% RSLogix 500 project IDENTIFICACION_BAK249.RSS, saved by version 7.30.00.17 %
PROJECT "UNTITLED"    % processor: MicroLogix 1500 %

PROGRAM FILES
  LAD 2 "PRINCIPAL"  5 rungs
  LAD 3 "FLUJO"  5 rungs
  LAD 4 "NIVEL"  9 rungs
  LAD 5 "BOMBAS"  5 rungs
  LAD 6 "FILTROS"  39 rungs

DATA FILES
  O0 OUTPUT  41 elements
  I1 INPUT  59 elements
  S2 STATUS  66 elements
  B3 BINARY  1 elements
  T4 TIMER  3 elements
  C5 COUNTER  1 elements
  R6 CONTROL  12 elements
  N7 INTEGER  84 elements
  F8 FLOAT  30 elements

LADDER 2 "PRINCIPAL"
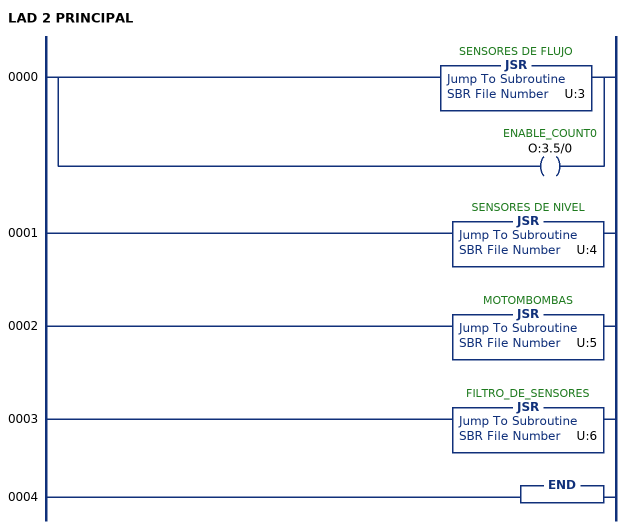
% Rung: 0 %
SOR BST JSR U:3 NXB OTE O:3.5/0 BND EOR
%   U:3  "SENSORES DE FLUJO" %
%   O:3.5/0  ENABLE_COUNT0 %
% Rung: 1 %
SOR JSR U:4 EOR
%   U:4  "SENSORES DE NIVEL" %
% Rung: 2 %
SOR JSR U:5 EOR
%   U:5  "MOTOMBOMBAS" %
% Rung: 3 %
SOR JSR U:6 EOR
%   U:6  FILTRO_DE_SENSORES %
% Rung: 4 %
SOR END EOR

LADDER 3 "FLUJO"
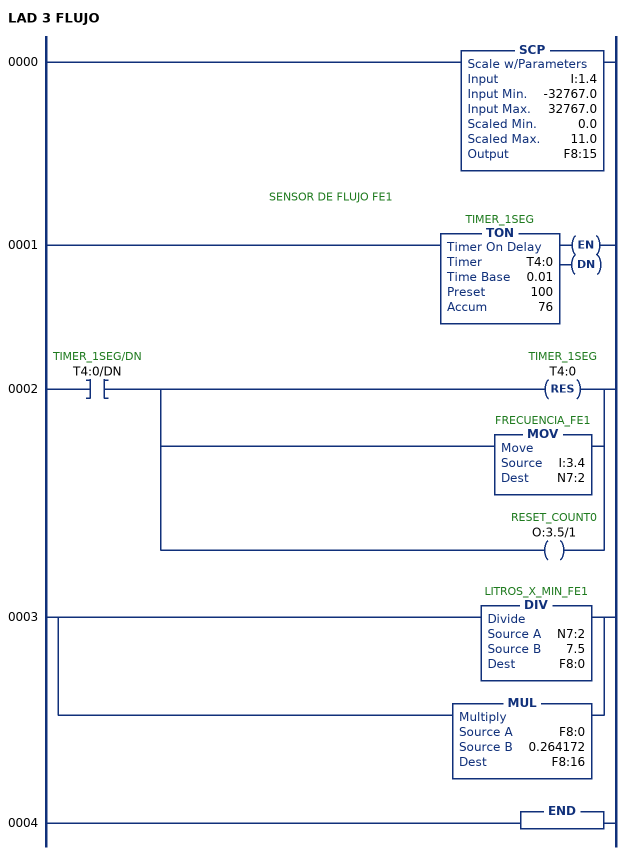
% Rung: 0 %
SOR SCP I:1.4 -32767.0 32767.0 0.0 11.0 F8:15 EOR
%   I:1.4  TRANSMISOR_FIT %
% Rung: 1 %
% SENSOR DE FLUJO FE1 %
SOR TON T4:0 0.01 100 76 EOR
%   T4:0  TIMER_1SEG %
% Rung: 2 %
SOR XIC T4:0/DN BST RES T4:0 NXB MOV I:3.4 N7:2 NXB OTE O:3.5/1 BND EOR
%   T4:0  TIMER_1SEG %
%   N7:2  FRECUENCIA_FE1 %
%   O:3.5/1  RESET_COUNT0 %
% Rung: 3 %
SOR BST DIV N7:2 7.5 F8:0 NXB MUL F8:0 0.264172 F8:16 BND EOR
%   N7:2  FRECUENCIA_FE1 %
%   F8:0  LITROS_X_MIN_FE1 %
% Rung: 4 %
SOR END EOR

LADDER 4 "NIVEL"
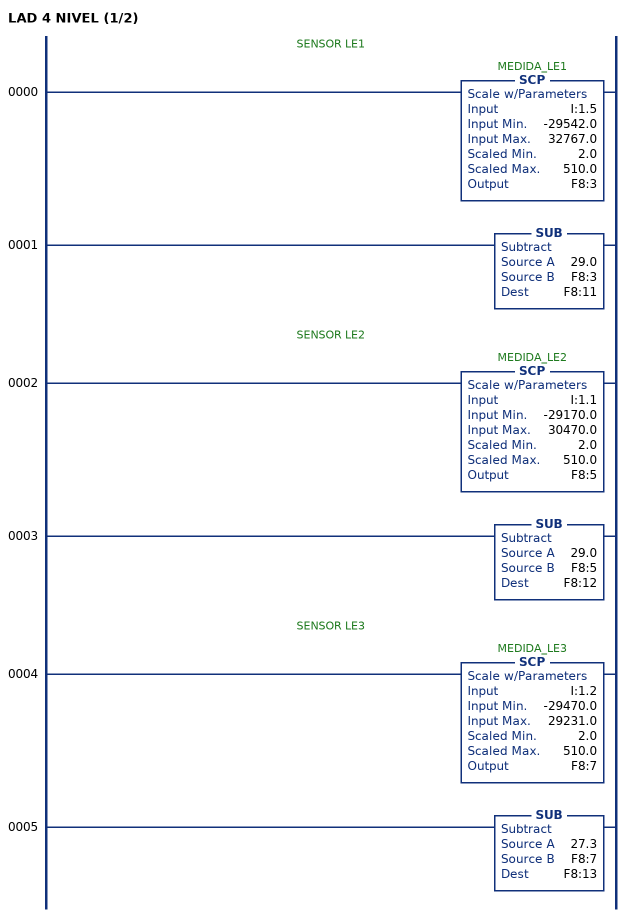
% Rung: 0 %
% SENSOR LE1 %
SOR SCP I:1.5 -29542.0 32767.0 2.0 510.0 F8:3 EOR
%   I:1.5  LE1 %
%   F8:3  MEDIDA_LE1 %
% Rung: 1 %
SOR SUB 29.0 F8:3 F8:11 EOR
%   F8:3  MEDIDA_LE1 %
% Rung: 2 %
% SENSOR LE2 %
SOR SCP I:1.1 -29170.0 30470.0 2.0 510.0 F8:5 EOR
%   I:1.1  LE2 %
%   F8:5  MEDIDA_LE2 %
% Rung: 3 %
SOR SUB 29.0 F8:5 F8:12 EOR
%   F8:5  MEDIDA_LE2 %
% Rung: 4 %
% SENSOR LE3 %
SOR SCP I:1.2 -29470.0 29231.0 2.0 510.0 F8:7 EOR
%   I:1.2  LE3 %
%   F8:7  MEDIDA_LE3 %
% Rung: 5 %
SOR SUB 27.3 F8:7 F8:13 EOR
%   F8:7  MEDIDA_LE3 %

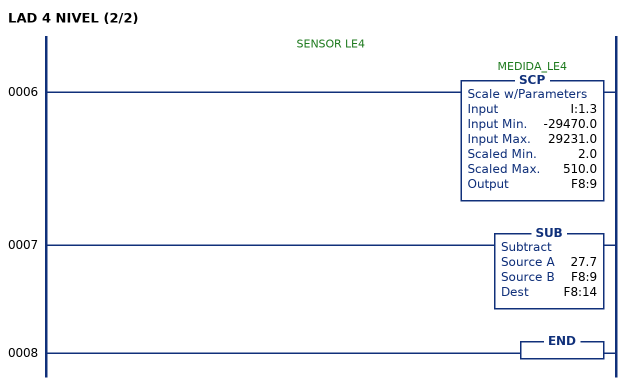
% Rung: 6 %
% SENSOR LE4 %
SOR SCP I:1.3 -29470.0 29231.0 2.0 510.0 F8:9 EOR
%   I:1.3  LE4 %
%   F8:9  MEDIDA_LE4 %
% Rung: 7 %
SOR SUB 27.7 F8:9 F8:14 EOR
%   F8:9  MEDIDA_LE4 %
% Rung: 8 %
SOR END EOR

LADDER 5 "BOMBAS"
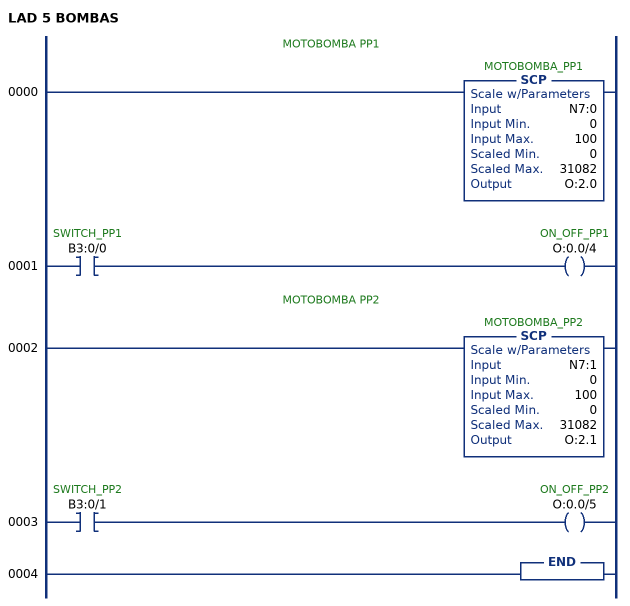
% Rung: 0 %
% MOTOBOMBA PP1 %
SOR SCP N7:0 0 100 0 31082 O:2.0 EOR
%   N7:0  FRECUENCIA_PP1 %
%   O:2.0  MOTOBOMBA_PP1 %
% Rung: 1 %
SOR XIC B3:0/0 OTE O:0.0/4 EOR
%   B3:0/0  SWITCH_PP1 %
%   O:0.0/4  ON_OFF_PP1 %
% Rung: 2 %
% MOTOBOMBA PP2 %
SOR SCP N7:1 0 100 0 31082 O:2.1 EOR
%   O:2.1  MOTOBOMBA_PP2 %
% Rung: 3 %
SOR XIC B3:0/1 OTE O:0.0/5 EOR
%   B3:0/1  SWITCH_PP2 %
%   O:0.0/5  ON_OFF_PP2 %
% Rung: 4 %
SOR END EOR

LADDER 6 "FILTROS"
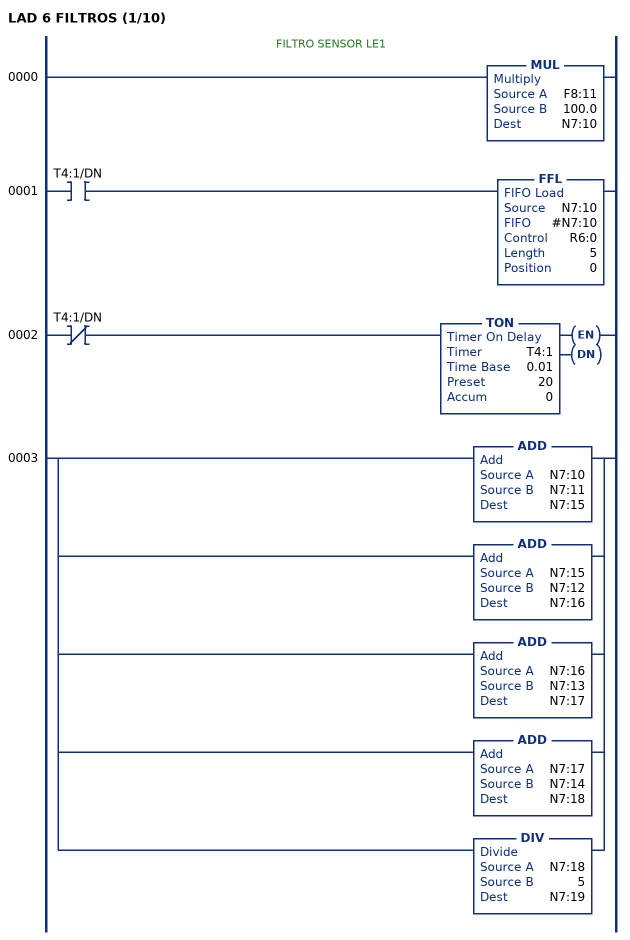
% Rung: 0 %
% FILTRO SENSOR LE1 %
SOR MUL F8:11 100.0 N7:10 EOR
% Rung: 1 %
SOR XIC T4:1/DN FFL N7:10 #N7:10 R6:0 5 0 EOR
% Rung: 2 %
SOR XIO T4:1/DN TON T4:1 0.01 20 0 EOR
% Rung: 3 %
SOR BST ADD N7:10 N7:11 N7:15 NXB ADD N7:15 N7:12 N7:16 NXB ADD N7:16 N7:13 N7:17 NXB ADD N7:17 N7:14 N7:18 NXB DIV N7:18 5 N7:19 BND EOR

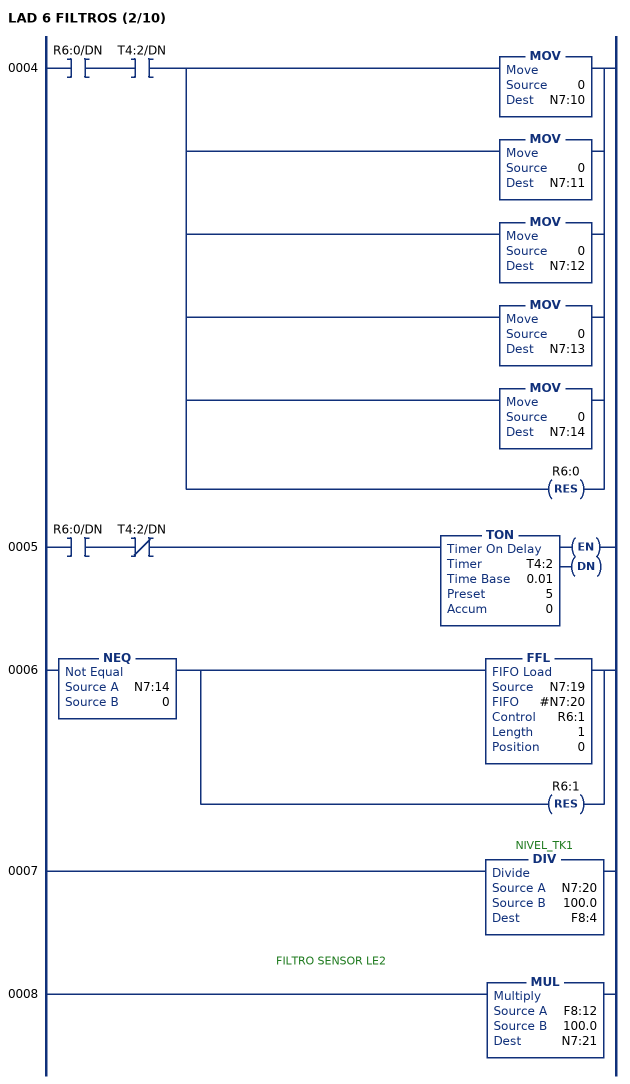
% Rung: 4 %
SOR XIC R6:0/DN XIC T4:2/DN BST MOV 0 N7:10 NXB MOV 0 N7:11 NXB MOV 0 N7:12 NXB MOV 0 N7:13 NXB MOV 0 N7:14 NXB RES R6:0 BND EOR
% Rung: 5 %
SOR XIC R6:0/DN XIO T4:2/DN TON T4:2 0.01 5 0 EOR
% Rung: 6 %
SOR NEQ N7:14 0 BST FFL N7:19 #N7:20 R6:1 1 0 NXB RES R6:1 BND EOR
% Rung: 7 %
SOR DIV N7:20 100.0 F8:4 EOR
%   F8:4  NIVEL_TK1 %
% Rung: 8 %
% FILTRO SENSOR LE2 %
SOR MUL F8:12 100.0 N7:21 EOR

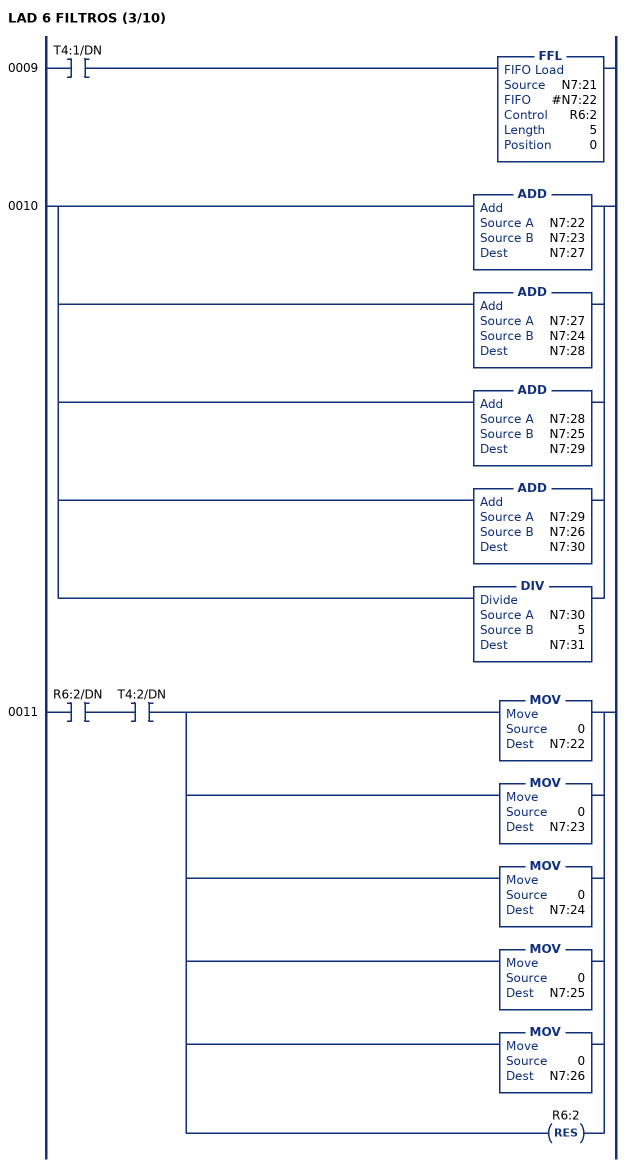
% Rung: 9 %
SOR XIC T4:1/DN FFL N7:21 #N7:22 R6:2 5 0 EOR
% Rung: 10 %
SOR BST ADD N7:22 N7:23 N7:27 NXB ADD N7:27 N7:24 N7:28 NXB ADD N7:28 N7:25 N7:29 NXB ADD N7:29 N7:26 N7:30 NXB DIV N7:30 5 N7:31 BND EOR
% Rung: 11 %
SOR XIC R6:2/DN XIC T4:2/DN BST MOV 0 N7:22 NXB MOV 0 N7:23 NXB MOV 0 N7:24 NXB MOV 0 N7:25 NXB MOV 0 N7:26 NXB RES R6:2 BND EOR

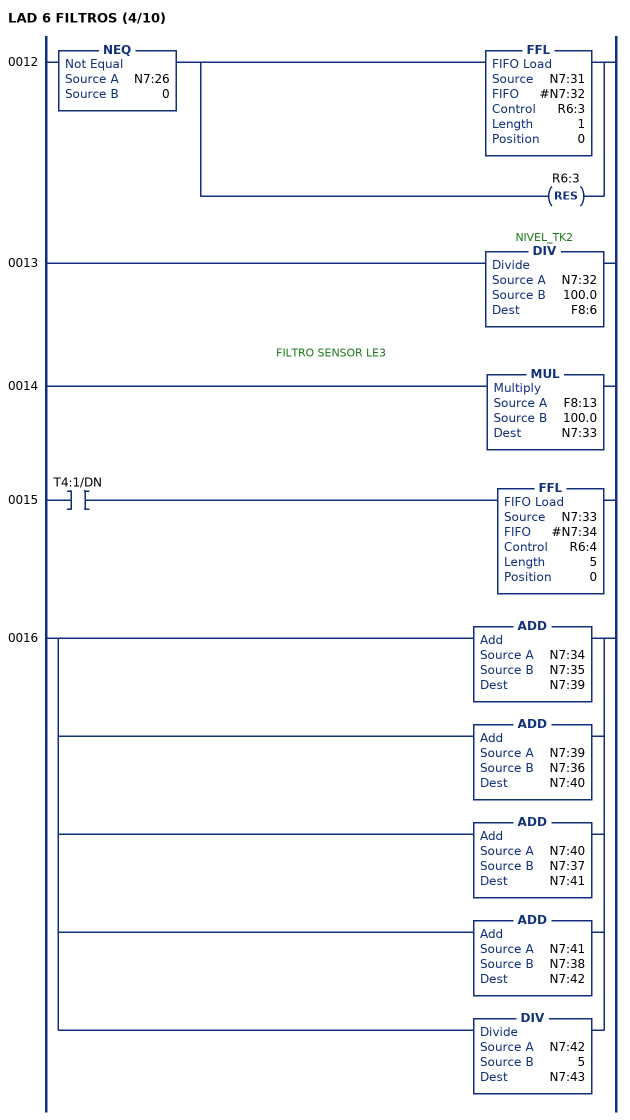
% Rung: 12 %
SOR NEQ N7:26 0 BST FFL N7:31 #N7:32 R6:3 1 0 NXB RES R6:3 BND EOR
% Rung: 13 %
SOR DIV N7:32 100.0 F8:6 EOR
%   F8:6  NIVEL_TK2 %
% Rung: 14 %
% FILTRO SENSOR LE3 %
SOR MUL F8:13 100.0 N7:33 EOR
% Rung: 15 %
SOR XIC T4:1/DN FFL N7:33 #N7:34 R6:4 5 0 EOR
% Rung: 16 %
SOR BST ADD N7:34 N7:35 N7:39 NXB ADD N7:39 N7:36 N7:40 NXB ADD N7:40 N7:37 N7:41 NXB ADD N7:41 N7:38 N7:42 NXB DIV N7:42 5 N7:43 BND EOR

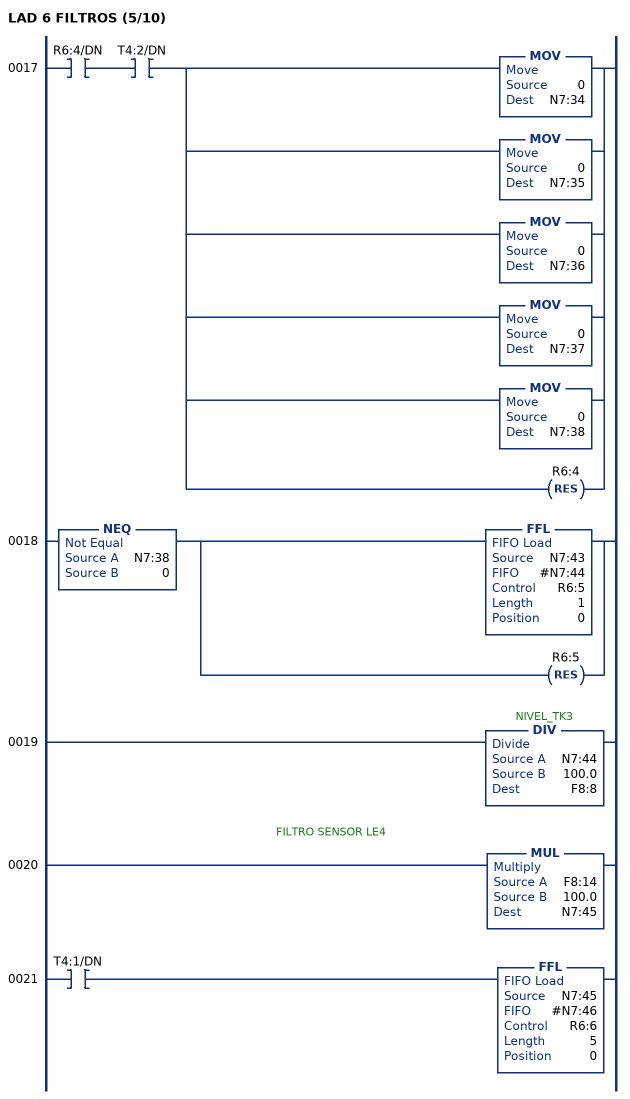
% Rung: 17 %
SOR XIC R6:4/DN XIC T4:2/DN BST MOV 0 N7:34 NXB MOV 0 N7:35 NXB MOV 0 N7:36 NXB MOV 0 N7:37 NXB MOV 0 N7:38 NXB RES R6:4 BND EOR
% Rung: 18 %
SOR NEQ N7:38 0 BST FFL N7:43 #N7:44 R6:5 1 0 NXB RES R6:5 BND EOR
% Rung: 19 %
SOR DIV N7:44 100.0 F8:8 EOR
%   F8:8  NIVEL_TK3 %
% Rung: 20 %
% FILTRO SENSOR LE4 %
SOR MUL F8:14 100.0 N7:45 EOR
% Rung: 21 %
SOR XIC T4:1/DN FFL N7:45 #N7:46 R6:6 5 0 EOR

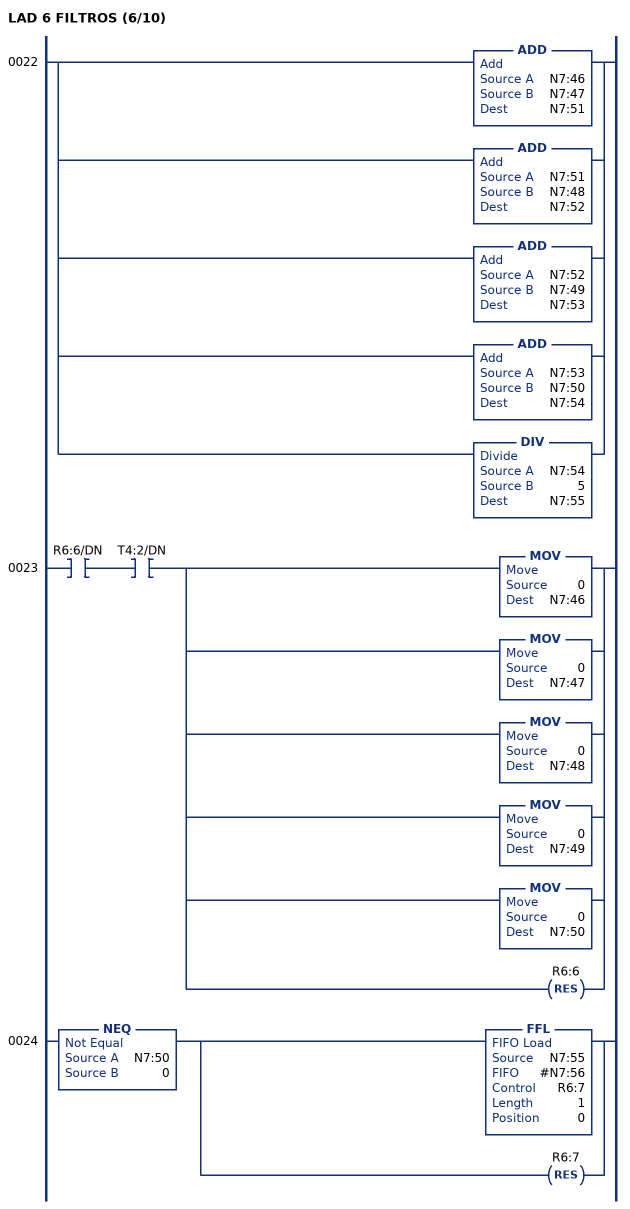
% Rung: 22 %
SOR BST ADD N7:46 N7:47 N7:51 NXB ADD N7:51 N7:48 N7:52 NXB ADD N7:52 N7:49 N7:53 NXB ADD N7:53 N7:50 N7:54 NXB DIV N7:54 5 N7:55 BND EOR
% Rung: 23 %
SOR XIC R6:6/DN XIC T4:2/DN BST MOV 0 N7:46 NXB MOV 0 N7:47 NXB MOV 0 N7:48 NXB MOV 0 N7:49 NXB MOV 0 N7:50 NXB RES R6:6 BND EOR
% Rung: 24 %
SOR NEQ N7:50 0 BST FFL N7:55 #N7:56 R6:7 1 0 NXB RES R6:7 BND EOR

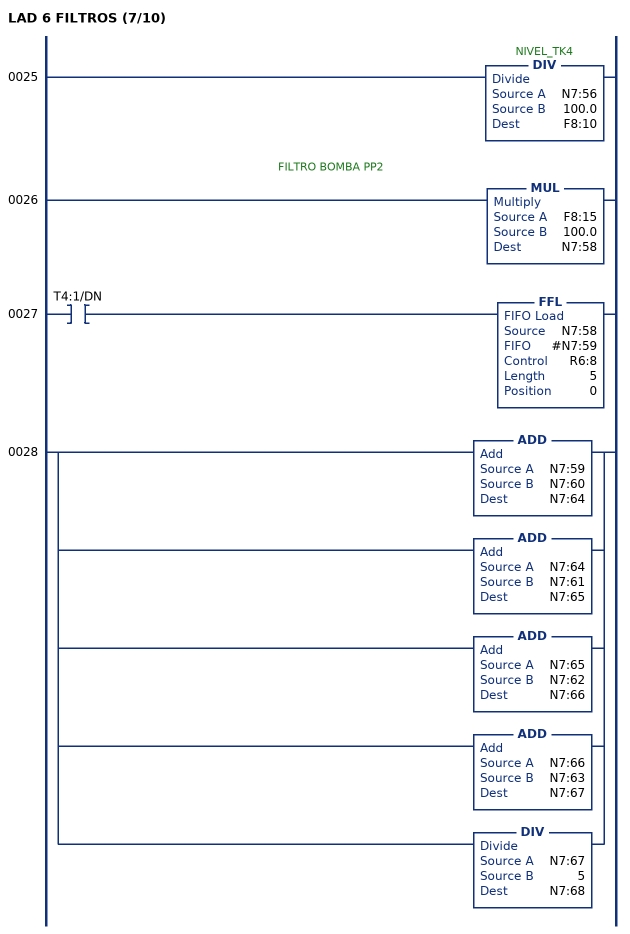
% Rung: 25 %
SOR DIV N7:56 100.0 F8:10 EOR
%   F8:10  NIVEL_TK4 %
% Rung: 26 %
% FILTRO BOMBA PP2 %
SOR MUL F8:15 100.0 N7:58 EOR
% Rung: 27 %
SOR XIC T4:1/DN FFL N7:58 #N7:59 R6:8 5 0 EOR
% Rung: 28 %
SOR BST ADD N7:59 N7:60 N7:64 NXB ADD N7:64 N7:61 N7:65 NXB ADD N7:65 N7:62 N7:66 NXB ADD N7:66 N7:63 N7:67 NXB DIV N7:67 5 N7:68 BND EOR

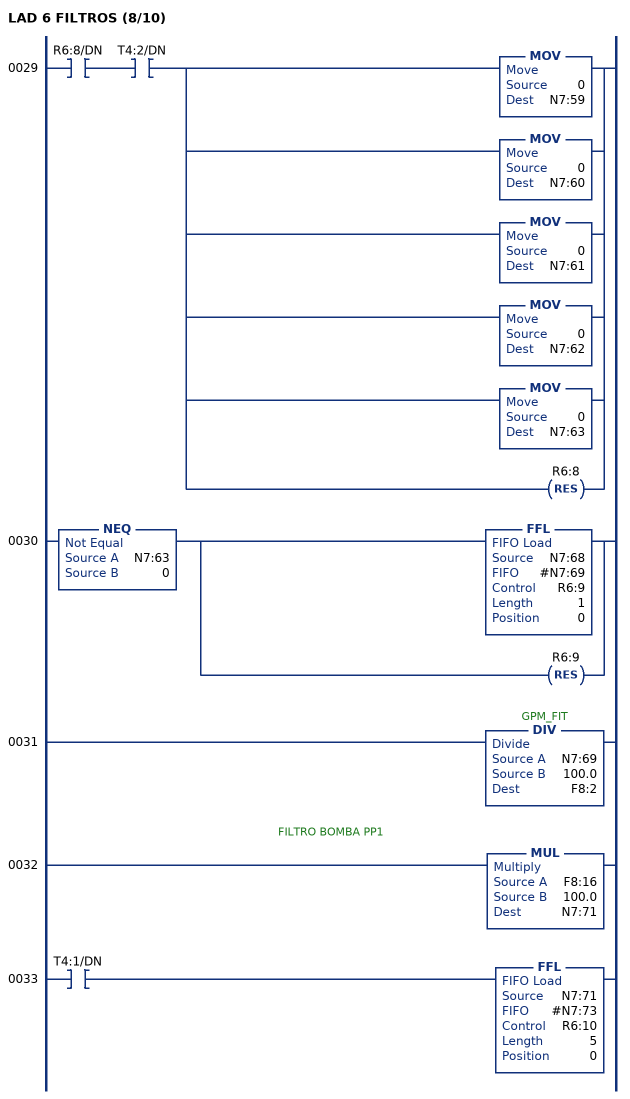
% Rung: 29 %
SOR XIC R6:8/DN XIC T4:2/DN BST MOV 0 N7:59 NXB MOV 0 N7:60 NXB MOV 0 N7:61 NXB MOV 0 N7:62 NXB MOV 0 N7:63 NXB RES R6:8 BND EOR
% Rung: 30 %
SOR NEQ N7:63 0 BST FFL N7:68 #N7:69 R6:9 1 0 NXB RES R6:9 BND EOR
% Rung: 31 %
SOR DIV N7:69 100.0 F8:2 EOR
%   F8:2  GPM_FIT %
% Rung: 32 %
% FILTRO BOMBA PP1 %
SOR MUL F8:16 100.0 N7:71 EOR
% Rung: 33 %
SOR XIC T4:1/DN FFL N7:71 #N7:73 R6:10 5 0 EOR

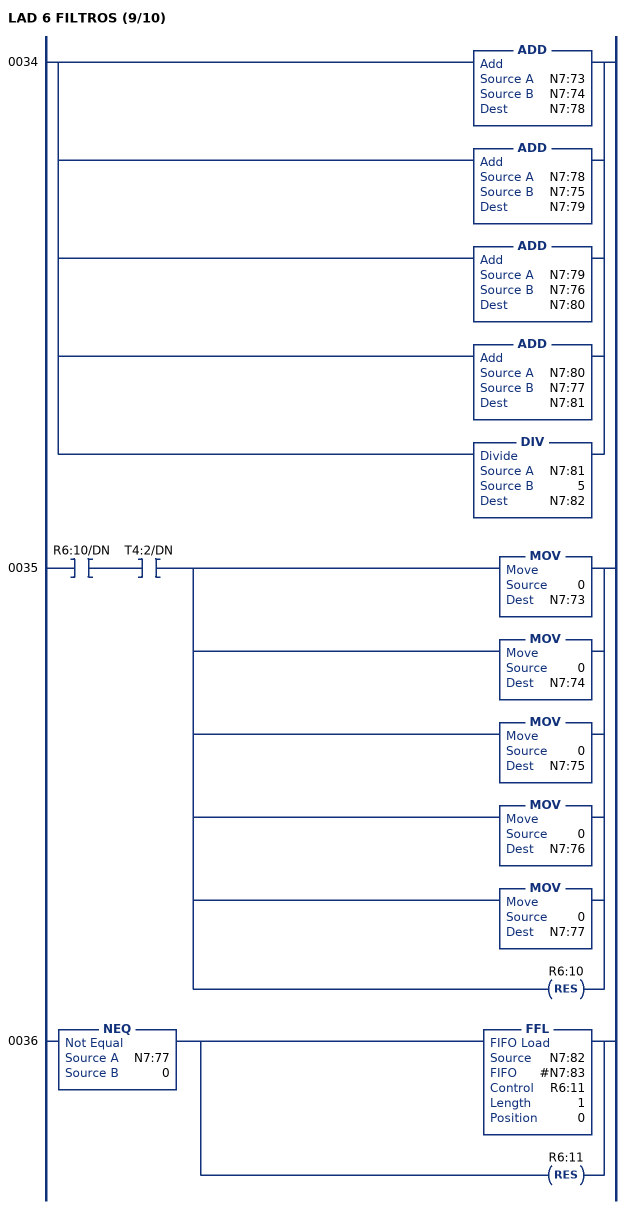
% Rung: 34 %
SOR BST ADD N7:73 N7:74 N7:78 NXB ADD N7:78 N7:75 N7:79 NXB ADD N7:79 N7:76 N7:80 NXB ADD N7:80 N7:77 N7:81 NXB DIV N7:81 5 N7:82 BND EOR
% Rung: 35 %
SOR XIC R6:10/DN XIC T4:2/DN BST MOV 0 N7:73 NXB MOV 0 N7:74 NXB MOV 0 N7:75 NXB MOV 0 N7:76 NXB MOV 0 N7:77 NXB RES R6:10 BND EOR
% Rung: 36 %
SOR NEQ N7:77 0 BST FFL N7:82 #N7:83 R6:11 1 0 NXB RES R6:11 BND EOR

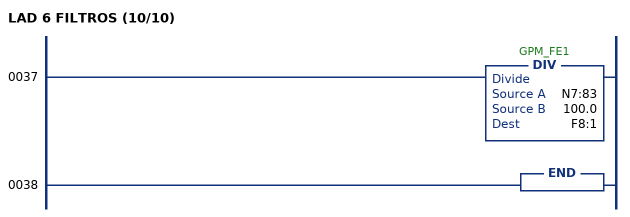
% Rung: 37 %
SOR DIV N7:83 100.0 F8:1 EOR
%   F8:1  GPM_FE1 %
% Rung: 38 %
SOR END EOR

COMMENTS NOT ATTACHED TO A CURRENT RUNG
  T9:0: PROMEDIO

DATA TABLE (non-zero values as saved)
DATA T4
% .PRE .ACC %
% T4:0 % 100 76
% T4:1 % 20 0
% T4:2 % 5 0
DATA C5
% .PRE .ACC %
% C5:0 % 15 0
DATA R6
% .LEN .POS %
% R6:0 % 5 0
% R6:1 % 1 0
% R6:2 % 5 0
% R6:3 % 1 0
% R6:4 % 5 0
% R6:5 % 1 0
% R6:6 % 5 0
% R6:7 % 1 0
% R6:8 % 5 0
% R6:9 % 1 0
% R6:10 % 5 0
% R6:11 % 1 0
DATA N7
% N7:0 % 100 100 0 0 0 0 0 0 0 0
% N7:10 % 0 0 0 0 19 0 0 0 0 0
% N7:20 % 0 1541 1490 0 0 0 0 0 0 0
DATA F8
% F8:0 % 0 162.2368 0.4975127 34.1714 -0.671402
% F8:5 % 27.09336 6.406641 33.80355 0.1964531 28.80152
% F8:10 % 5.698481 0 0 0 0
% F8:15 % 0.4948271 0 0 0 0
